FUNCTION fAnalogSensorScale : INT
VAR_INPUT
	IN:INT;
	ptr:POINTER TO AnalogSensorCalibrationTyp;
END_VAR
VAR
	M:REAL;
	B:REAL;
	TEMPX:REAL;
END_VAR

TEMPX := (ptr^.X2-ptr^.X1);
IF TEMPX<>0 THEN
	M:=(ptr^.Y2-ptr^.Y1)/(ptr^.X2-ptr^.X1);
END_IF

IF ptr^.X1 <> 0 AND M <>0 THEN
	B:= ptr^.Y1-(M*ptr^.X1);
	fAnalogSensorScale := REAL_TO_INT(M*IN+B);
ELSIF ptr^.X2 <> 0 AND M <>0 THEN
	B:= ptr^.Y2-(M*ptr^.X1);
	fAnalogSensorScale := REAL_TO_INT(M*IN+B);
END_IF

END_FUNCTION

(* stored: Version 1.1.0.1, ProductVersion 3.1.4024.3
   POU fAnalogSensorScale: Id {b49c3e14-8a54-0eed-1294-d2245bd9a653}, SpecialFunc None *)
